TYPE Valj :
STRUCT
	id: INT;
	pos: POZICIJA;
END_STRUCT
END_TYPE

(* stored: Version 1.1.0.1, ProductVersion 3.1.4024.12
   DUT Valj: Id {a6aafdbd-5312-4569-b8f4-74d9ff70f972} *)
